PROGRAM MAIN
VAR

	// ========= System Control / FSM Variables =========
	
	MainCommands 		: MainCommands_typ; 	// command struct for cycling thru the state machine
	MainState    		: MainState_enum;   	// enumeration for the Main state machine

	// ========= Linked NC Variables & References =========
	
	Mover    			: ARRAY[0..GVL.NUM_MOVERS - 1] OF Mover; 	// instantiation of Mover objects. Matches the number of movers on the system
    GroupRef 			: AXES_GROUP_REF;                       	 // linked to the Collision Avoidance group and passed cyclically to every Mover object

	// ========= Objectives & Parameters =========

    MoverList    		: MoverList;
    ParameterSet 		: MotionParameters_typ;

    Station         	: ARRAY[0..GVL.NUM_STATIONS - 1] OF Station;
    PositionTrigger 	: ARRAY[0..2] OF PositionTrigger;
    SpeedTrigger    	: ARRAY[0..1] OF SpeedTrigger;
    Zone            	: ARRAY[0..3] OF Zone;
	
    // ========= Example Application Variables =========

    nextStation 		: USINT := 4;
                    	
    lowVelocity    		: LREAL := 200;  	// mm/s
    mediumVelocity 		: LREAL := 800;  	// mm/s
    highVelocity   		: LREAL := 1200; 	// mm/s

    // ========= Helper, State, & Index Variables =========
	
    i                	: UINT; 	// index variable; gets reused in various FOR loops
    n                	: UINT; 	// secondary index variable, for enabling movers
    allMoversEnabled 	: BOOL; 	// helper flag for verifying enable status of all movers
	allMoverTracksEnabled : BOOL;	// helper flag for verifying track active status of all movers
	allMoversDisabled	: BOOL;		// helper flag for verifying disable status of all movers
	allMoversHalted		: BOOL;		// helper flag for verifying halt status of all movers

    StationTimer 		: ARRAY[0..GVL.NUM_STATIONS] OF TON; // timer blocks, for station dwells	
	
	// ========= XTS Utility Diagnostics =========
	
	VisuDiag						: FB_VisuXtsDiag;
	fbXtsEnvironment				: FB_TcIoXtsEnvironment;
	fbXtsEnvironmentVisu			: FB_XtsEnvironmentVisu;
	stXtsEnvironmentConfiguration	: ST_XtsEnvironmentConfiguration;
	nEnvironmentState				: INT;
	
	// ======== Track management ========
	Track		: ARRAY [0..GVL.NUM_TRACKS] OF Track;
	
	
	// ======== Queue Logic Variables ========
	temp_payload : payload_TYP;
	SB_dispensers : ARRAY [1..3] OF StarburstDispenser;
	//make an array
	
	
	current_order : Order_TYP;
	hmi_order : Order_TYP;
	red : INT;
	orange : INT;
	pink : INT;
	bconfirm_order: BOOL := FALSE;
	bpicked_up: BOOL;
	
	order_num_signal: INT;
	temp: Payload_TYP;
END_VAR

	



(* ======================================================================================

--- XTS Starter Project ---

This MAIN (PRG) is intended to serve as an example, which can be modified to suit your specific application.

No programming changes should be necessary inside the provided XTS objects / function block definitions.
They are intended to be simply instantiated and controlled via the provided methods and properties.
However the objects are provided as open-source for modification and extension as needed.

Documentation for these objects can be found online at:
https://beckhoff-usa-community.github.io/XTS_Base/

Bug reports, new feature requests, and general feedback is always welcome on our Github page.
For any other questions, please reach out to your local Application Engineer.

- Beckhoff USA Advanced Applications Group

====================================================================================== *)





CASE MainState OF
    MS_DISABLED: // --------------------------------------------------------- IDLE STATE
		(*Wait here until an operator issues a MainCommand to Enable the system. 
		Disallow Start and Stop commands until the system has been Enabled*)
	
        MainCommands.Start		:= FALSE;
		MainCommands.Stop		:= FALSE;
		
        IF MainCommands.Enable THEN
            MainCommands.Disable := FALSE;
            MainState            := MS_INITIALIZING_MOVERS;
        END_IF

    MS_INITIALIZING_MOVERS: // --------------------------------------------- SET MOVER MOTION PARAMETERS
		(*Initialize Mover motion parameters via a Parameter Set. Once complete, step
		forward to begin Enabling movers on the system*)
		
		ParameterSet.Jerk         := 1E5; // mm/s3
		ParameterSet.Acceleration := 1E4; // mm/s2
		ParameterSet.Deceleration := 1E4; // mm/s2
		ParameterSet.Velocity     := 1E3; // mm/s
		ParameterSet.Direction    := mcDirectionPositive;

        FOR i := 0 TO GVL.NUM_MOVERS - 1 DO
            Mover[i].MotionParameters := ParameterSet;
        END_FOR
		
		IF MainCommands.Disable THEN
			MainCommands.Enable		:= FALSE;
			MainState				:= MS_DISABLED;
		ELSIF MainCommands.Stop THEN
			MainCommands.Stop		:= FALSE;
			MainCommands.Disable	:= TRUE;
			MainCommands.Start		:= FALSE;
			MainState				:= MS_DISABLED;
		ELSIF MainCommands.Enable THEN
        	MainState 				:= MS_ONESHOT_ENABLE;
		END_IF

	MS_ONESHOT_ENABLE:	// -------------------------------------------------- SINGLE-CYCLE ISSUE ENABLE COMMANDS
		(*Begin Enabling movers by calling Mover.Enable(). Methods in this project
		are intended to be called once, although they will function correctly if called repeatedly*)

		FOR i := 0 TO GVL.NUM_MOVERS - 1 DO
			Mover[i].Enable();
		END_FOR

		MainState		:= MS_ENABLING_MOVERS;
	
    MS_ENABLING_MOVERS: // -------------------------------------------------- RESETTING AND ENABLING AXES
		(*Wait here until all movers have Enabled. This means that the Axis has
		fully energized, and also that all Collision Avoidance grouping and Mover 1 detection
		has finished. If the state machine gets stuck in this state, check the Error output
		of an individual Mover to see what the issue is. A common cause is forgetting to link
		Mover NC Axes to the AXIS_REF inside the PLC*)

        allMoversEnabled := TRUE; // default ...

        FOR i := 0 TO GVL.NUM_MOVERS - 1 DO
            IF Mover[i].Ready = FALSE THEN
                allMoversEnabled 		:= FALSE;
            END_IF
        END_FOR

        IF allMoversEnabled THEN
			IF MainCommands.Disable THEN
				MainCommands.Enable		:=FALSE;
            	MainState				:= MS_ONESHOT_DISABLE;
			ELSIF MainCommands.Stop	 THEN
				MainCommands.Start		:=FALSE;
				MainState				:= MS_ONESHOT_STOP;
			ELSIF MainCommands.Enable THEN
	        	MainState 				:= MS_INITIALIZING_OBJECTIVES;
			END_IF
        END_IF

    MS_INITIALIZING_OBJECTIVES: // --------------------------------------------- WRITING OBJECTIVE PARAMETERS
		(*Initialize Station positions, Position Trigger positions, Zones etc. *)

        // Initialize station positions
        Station[0].Position := 1250;
        Station[1].Position := 25;
        Station[2].Position := 127;
        Station[3].Position := 228;
        Station[4].Position := 875;

       
        Zone[0].StartPosition := 0;
        Zone[0].EndPosition   := 1500;

		
		// give all tracks their ID number
		FOR i := 0 TO GVL.NUM_TRACKS DO
			Track[i].Id := UINT_TO_INT(i);
		END_FOR
		
		// Track 0 is a special case absolute reference, no-modulus track instance and is not normally used
		Track[0].OTCID := 0;				// special "absolute reference" case
		Track[1].OTCID:= 16#01010290;		// value copied from XtsProcessingUnit1 > Track x > Object > Object Id field

		MainState := MS_ACTIVATE_TRACKS;
		
	MS_ACTIVATE_TRACKS:
		// activate all movers on track[1]
		FOR i := 0 TO GVL.NUM_MOVERS - 1 DO
            Mover[i].ActivateTrack(Track[1]);
        END_FOR
		
		MainState := MS_WAIT_FOR_TRACKS;
	
	MS_WAIT_FOR_TRACKS:
		// wait for all movers to activate their tracks
		
		allMoverTracksEnabled := TRUE;
		FOR i := 0 TO GVL.NUM_MOVERS - 1 DO
			IF (NOT Mover[i].IsTrackReady) THEN
            	allMoverTracksEnabled := FALSE;
			END_IF;
        END_FOR
		IF (allMoverTracksEnabled) THEN
			MainState := MS_ENABLED;	
		END_IF

    MS_ENABLED: // ------------------------------------------------------------- MOVERS ENABLED, STOPPED
		(*In this state, Movers should be energized and holding their position. They should wait
		until a Start command is issued. This is also a good state to include basic Recovery steps.
		Our example shows a simple use-case involving Zones for localized recovery*)

		MainCommands.Stop	:= FALSE;
	
        IF MainCommands.Start THEN

            // ===== RECOVERY LOGIC =====

            (*
			Recovery is typically very application-specific. Each implementation will need to determine
			what to do with work-in-progres, rejects, movers with unknown product status, etc.s
			*)

            // Register all movers with all Zones, for recovery
            FOR i := 0 TO GVL.NUM_MOVERS - 1 DO
                Zone[0].RegisterMover( Mover[i] );
            END_FOR
			
            Zone[0].CurrentMoverList.SetAllVelocity(200).MoveAllToStation(Station[0]);

            // ===== END =====

            MainState			:= MS_RUN;

        ELSIF MainCommands.Disable THEN
            MainCommands.Enable := FALSE;
            MainState           := MS_ONESHOT_STOP;
        END_IF

    MS_RUN: // --------------------------------------------------------------- OPERATING
		(*Mover routing logic should be written here to define the system's operating behavior.
		Station implementations, Position Trigger logic, etc. In general, you can remove the example code
		here down to the short line break that looks like this: // ============= *)
	
	
		// Recieves order from user and populates queue
		IF bconfirm_order THEN
			hmi_order.order_num := GVL.order_number;
			hmi_order.red := red;
			hmi_order.orange := orange;
			hmi_order.pink := pink;
			GVL.order_number := GVL.order_number + 1;
			
			//enqueues order
			Orders.ENQUEUE(hmi_order);
			// sets temporary variable holding the order information for the mover
			current_order := Orders.order;
			bconfirm_order := FALSE;
		END_IF
		
		
	
		
        // Station 0 Logic for start station
        IF Station[0].MoverInPosition THEN
			
			//Check if there is an order available
			IF Orders.HasOrder THEN
				
				//delete order off of the queue
				Orders.DEQUEUE();
	
				
			
				//set mover payload with order info
				temp_payload := Station[0].CurrentMover.Payload;
				temp_payload.Red := current_order.red;
				temp_payload.Orange := current_order.orange;
				temp_payload.Pink := current_order.pink;
				temp_payload.Order_Num := current_order.order_num;
				Station[0].CurrentMover.Payload := temp_payload;
				
				//Move to first station
				Station[0].CurrentMover.SetVelocity(500);
                Station[0].CurrentMover.MoveToStation(Station[1]);
				
				
			END_IF
       END_IF
		
        // Station 1 Logig for Red starbursts	
        IF Station[1].MoverInPosition THEN
			
			// dispenses red starbursts
			SB_dispensers[1](mover := Station[1].currentMover, station_num := 1, dispense := TRUE);
			
			//when done dispensing mover goes to next station
			IF SB_dispensers[1].completed THEN;
				SB_dispensers[1](mover := Station[1].currentMover, station_num := 1, dispense := FALSE);
                Station[1].CurrentMover.SetVelocity(500);
                Station[1].CurrentMover.MoveToStation(Station[2]);
            END_IF
			
        END_IF
		
		//Station 2 logic for Orange starbursts
		IF Station[2].MoverInPosition THEN
            
			// dispenses orange starbursts
			SB_dispensers[2](mover := Station[2].currentMover, station_num := 2, dispense := TRUE);
			
			//when done dispensing mover goes to next station
			IF SB_dispensers[2].completed THEN
                Station[2].CurrentMover.SetVelocity(500);
                Station[2].CurrentMover.MoveToStation(Station[3]);
				SB_dispensers[2](mover := Station[2].currentMover, station_num := 2, dispense := FALSE);
            END_IF
  
        END_IF
		
		
		
		//Station 3 logic for Pink starbursts
		IF Station[3].MoverInPosition THEN
			
			//dispense pink starbursts
			SB_dispensers[3](mover := Station[3].currentMover, station_num := 3, dispense := TRUE);
			
			//when done dispensing mover goes to next station
			IF SB_dispensers[3].completed THEN
                Station[3].CurrentMover.SetVelocity(500);
                Station[3].CurrentMover.MoveToStation(Station[4]);
				SB_dispensers[3](mover := Station[3].currentMover, station_num := 3, dispense := FALSE);
            END_IF
			
        END_IF
		
		
		
		//Station 4 logic for pickup station
		IF Station[4].MoverInPosition THEN
            
			temp := Station[4].CurrentMover.Payload;
			order_num_signal := temp.Order_Num;
			
		
			// Once picked up, move back to starting station
            IF bpicked_up THEN
				
				// Ping signal to Orders.queue[Orders.first_order] for that order_num
                Station[4].CurrentMover.SetVelocity(1000);
                Station[4].CurrentMover.MoveToStation(Station[0]);
            END_IF
       
        END_IF
		
		
	
		// Example call to XTS Utility library. See Diagnostics section of docs for more info
		(*
		myMoverMileage	:= fbXtsEnvironment.XpuTcIo(1).MoverTcIo(2).GetDistanceDriven();
		*)
		
		// =============

        IF MainCommands.Stop THEN
            MainCommands.Start 	:= FALSE;
            MainState         	:= MS_ONESHOT_STOP;
        ELSIF MainCommands.Disable THEN
            MainCommands.Enable := FALSE;
            MainState           := MS_ONESHOT_STOP;
        END_IF
		
	MS_ONESHOT_STOP:	// --------------------------------------------------- SINGLE-CYCLE ISSUE HALT COMMANDS
		(*Issue a halt command, then change states right away to wait for Movers to carry out the instruction*)
	
		FOR i := 0 TO GVL.NUM_MOVERS - 1 DO
			Mover[i].Halt();
		END_FOR
	
		MainState					:= MS_STOPPING;
	
    MS_STOPPING: // ---------------------------------------------------------- STOPPING MOVERS
		(*Movers are coming to a stop here in this state*)

		// Stop all movers
		allMoversHalted				:= TRUE;
		FOR i := 0 TO GVL.NUM_MOVERS - 1 DO
			Mover[i].AxisReference.ReadStatus();
			IF Mover[i].AxisReference.Status.Moving THEN
				allMoversHalted		:= FALSE;
			END_IF
		END_FOR
		
		MainCommands.Start			:= FALSE;
 
		IF allMoversHalted THEN
           	MainState 				:= MS_STOPPED;
		END_IF
        

    MS_STOPPED: // ------------------------------------------------------------ Stop Command has been sent, hold here
		(*Movers are now stopped, and further Main Commands can be issued to the system*)

        IF MainCommands.Disable THEN
            MainCommands.Enable 	:= FALSE;
			MainCommands.Start		:= FALSE;
            MainState           	:= MS_ONESHOT_DISABLE;
        ELSIF MainCommands.Start THEN
            MainCommands.Stop 		:= FALSE;
            MainState         		:= MS_ENABLING_MOVERS;
        END_IF

	    // Reinit nextStation
        nextStation := 4;

        // Unregister everything from all stations
        FOR i := 0 TO GVL.NUM_STATIONS - 1 DO
            Station[i].UnregisterAll();
        END_FOR

        // Unregister everything from all Pos Trigs
        FOR i := 0 TO SIZEOF(PositionTrigger) / SIZEOF(PositionTrigger[0]) - 1 DO
            PositionTrigger[i].UnregisterAll();
        END_FOR

        // Unregister everything from all speed trigs
        FOR i := 0 TO SIZEOF(SpeedTrigger) / SIZEOF(SpeedTrigger[0]) - 1 DO
            SpeedTrigger[i].UnregisterAll();
        END_FOR

        // Unregister everything from all zones
        FOR i := 0 TO SIZEOF(Zone) / SIZEOF(Zone[0]) - 1 DO
            Zone[i].UnregisterAll();
        END_FOR
	
	MS_ONESHOT_DISABLE:	// ------------------------------------------------------- SINGLE CYCLE ISSUE DISABLE COMMANDS
		(*Mover disable commands are issued here, followed by a state tranisition to await completion of the Disabling*)
		FOR i := 0 TO GVL.NUM_MOVERS DO
			Mover[i].Disable();
		END_FOR

		MainState					:=	MS_DISABLING;
	
    MS_DISABLING: // --------------------------------------------------- DISABLING MOVERS
		(*Movers are Disabling. During this step, we also Unregister movers from relevant Objectives
		to ensure proper startup behavior*)
		
        // Reinit nextStation
        nextStation := 4;

        // Unregister everything from all stations
        FOR i := 0 TO GVL.NUM_STATIONS - 1 DO
            Station[i].UnregisterAll();
        END_FOR

        // Unregister everything from all Position triggers
        FOR i := 0 TO SIZEOF(PositionTrigger) / SIZEOF(PositionTrigger[0]) - 1 DO
            PositionTrigger[i].UnregisterAll();
        END_FOR

        // Unregister everything from all speed triggers
        FOR i := 0 TO SIZEOF(SpeedTrigger) / SIZEOF(SpeedTrigger[0]) - 1 DO
            SpeedTrigger[i].UnregisterAll();
        END_FOR

        // Unregister everything from all zones
        FOR i := 0 TO SIZEOF(Zone) / SIZEOF(Zone[0]) - 1 DO
            Zone[i].UnregisterAll();
        END_FOR
		
		allMoversDisabled				:= TRUE;
		
		FOR i := 0 TO gvl.NUM_MOVERS-1 DO
			IF NOT Mover[i].AxisReference.Status.Disabled THEN 
				allMoversDisabled		:= FALSE;
			END_IF
		END_FOR
 
        IF allMoversDisabled THEN
            MainState					:= MS_DISABLED;
        END_IF

    MS_ERROR: // --------------------------------------------------- ERRORSTATE
		(*A reset command can be included here to clear Mover errors, etc. and return
		to a controlled state*)

    MS_DEBUG: // ------------------------------------------------------- DEV USE ONLY
		(*This state is intentionally left blank, 
		for optional use by a developer during programming*)
	

END_CASE;

// Initialize and update diagnostic features
InitializeUtilityLibrary();

// Call all mover function blocks cyclically
FOR i := 0 TO GVL.NUM_MOVERS - 1 DO
    Mover[i].Cyclic(GroupRef);
	Mover[i].AxisReference.ReadStatus();
END_FOR;

// Call all station function blocks cyclically
FOR i := 0 TO GVL.NUM_STATIONS - 1 DO
    Station[i].Cyclic();
END_FOR

// Call trigger function blocks cyclically
PositionTrigger[0].Cyclic();
PositionTrigger[1].Cyclic();
PositionTrigger[2].Cyclic();

SB_dispensers[1]();
SB_dispensers[2]();
SB_dispensers[3]();

ACTION InitializeUtilityLibrary:



CASE nEnvironmentState OF
	0:	// ----------------------------------------- Enable Init Items
	
		// Enable init Info Server if needed
		stXtsEnvironmentConfiguration.bEnableInitInfoServer		:= TRUE;
		
		// Enable init CA Group if needed
		stXtsEnvironmentConfiguration.bEnableInitCaGroup		:= TRUE;
		
		// Set configuration of XtsUtility init
		fbXtsEnvironment.P_XtsEnvironmentConfiguration			:= stXtsEnvironmentConfiguration;
		
		// Next step
		nEnvironmentState	:= 1;
		
	1:	// ------------------------------------------ Init Environment
		
		// Start init
		IF fbXtsEnvironment.Init(TRUE) THEN
			// stop init
			fbXtsEnvironment.Init(FALSE);
			
			// next step
			nEnvironmentState	:= 2;
		END_IF
		
	2:	// ------------------------------------------ Check for success
	
		// Check IsInitialized property
		IF fbXtsEnvironment.P_IsInitialized THEN
			// next step
			nEnvironmentState	:= 3;
		END_IF
		
	3:	// ------------------------------------------- Init Visu
	
		fbXtsEnvironmentVisu( ipTcIoXtsEnvironment := fbXtsEnvironment );
		
		// next step
		nEnvironmentState	:= 4;
		
	4:	// ------------------------------------------- Init done

		fbXtsEnvironmentVisu.Cycle();
		
END_CASE
END_ACTION

END_PROGRAM

(* stored: Version 1.1.0.1, ProductVersion 3.1.4024.13
   POU MAIN: Id {0790caa7-8a3f-4f91-b0f8-9ebb3db3858d}, SpecialFunc None
   Action InitializeUtilityLibrary: Id {4ac3b602-bbee-0af7-24db-b9d89bbd3ae5} *)
